SUBAPPLICATION Ventilsteuerung_Uebung_034a1_Q2 (* Numeric Value Input auf PWM Ausgang *)
  (* Standard: 61499-2 *)
  (* Version 1.0, 2023-10-23, franz *)
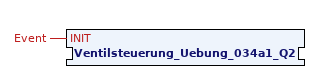
  EVENT_INPUT
    INIT;
  END_EVENT
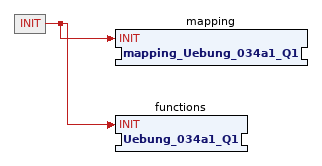
  SUBAPPS
    mapping : mapping_Uebung_034a1_Q1;
    functions : Uebung_034a1_Q1;
  END_SUBAPPS
  EVENT_CONNECTIONS
    INIT TO mapping.INIT;
    INIT TO functions.INIT;
  END_CONNECTIONS
END_SUBAPPLICATION
